FUNCTION Between : BOOL // Returns true if value is >= the lower and <= the upper threshold
VAR_INPUT
	Lower	: LREAL	; // lower threshold value [LREAL]
	Value	: LREAL	; // test value [LREAL]
	Upper	: LREAL	; // Upper threshold value [LREAL]
END_VAR
VAR
END_VAR

// Check if value is between lower and upper threshold
Between := (Value >= Lower) AND (Value <= Upper);

END_FUNCTION

(* stored: Version 1.1.0.1, ProductVersion 3.1.4024.3
   POU Between: Id {636b1549-e7ce-4101-8455-6287d049e510}, SpecialFunc None *)
